(* PLC project Tc3_EventLogger.ipSourceInfo Demo, tc3-libraries-kb TwinCAT 3.1 *)
(* stored: creationDateTime 2026-05-11T01:00:00, modificationDateTime 2026-05-11T01:00:00 *)

PROGRAM P_Demo_ipSourceInfo
  VAR
    fbAlarm : FB_TcAlarm;  (* alarm 实例（已 Create） *)
    ipSrc : I_TcSourceInfo;  (* 源信息接口 *)
    sSourceName : STRING;  (* 拿到的 SourceName *)
  END_VAR

// =============================================================================
// 场景：读取 alarm 的源信息用于日志归档
// 价值：一次调用拿到 SourceInfo 接口供后续读 SourceName/SourceID
// 验证：登录后 monitor ipSrc，应能拿到非 0 接口；调用 ipSrc 上的 getter 能读出 SourceName 字符串
// 验证步骤：
//   1. 右键 PLC 项目 → Import PLCopenXML → 选本文件
//   2. 引用 Tc3_EventLogger（System → References → Add library）
//   3. 编译 → 登录 → 运行；按 verify 注释里给出的在线写值操作
// =============================================================================

ipSrc := fbAlarm.ipSourceInfo;
IF ipSrc &lt;&gt; 0 THEN
    sSourceName := ipSrc.sSourceName;     // I_TcSourceInfo 的属性
END_IF;
END_PROGRAM
